FUNCTION_BLOCK CsvPersistantEventStorage IMPLEMENTS I_PersistentEventStorage
VAR
	fbFileOpen : FB_FileOpen := (sPathName := 'C:\Events.log', nMode := FOPEN_MODEAPPEND OR FOPEN_MODETEXT);
	fbFilePuts : FB_FilePuts;
	fbFileClose : FB_FileClose;
	eWriteState : (FILE_OPEN_TRIGGER,FILE_OPEN, WAIT_FOR_EVENT,WRITE_EVENT_TRIGGER, WRITE_EVENT, FILE_CLOSE_TRIGGER, FILE_CLOSE, ERROR);
	stEventWrittenToFile : ST_Event;
	CsvString: T_MaxString;
END_VAR

CASE eWriteState OF
	FILE_OPEN_TRIGGER :
		fbFileOpen(bExecute := TRUE);
		
	FILE_OPEN :
		fbFileOpen(bExecute := FALSE);
		IF fbFileOpen.bError THEN
			eWriteState := ERROR;
		ELSIF NOT fbFileOpen.bBusy AND fbFileOpen.hFile <> 0 THEN
			eWriteState := WAIT_FOR_EVENT;
		END_IF
		
	WAIT_FOR_EVENT : 
		// Do nothing
		
	WRITE_EVENT_TRIGGER : 
		CsvString := CreateCsvString(stEvent := stEventWrittenToFile);
		fbFilePuts(bExecute := TRUE,
			sLine := CsvString,
			hFile := fbFileOpen.hFile);
		eWriteState := WRITE_EVENT;
		
	WRITE_EVENT :
		fbFilePuts(bExecute := FALSE);
		IF fbFilePuts.bError THEN
			eWriteState := ERROR;
		ELSIF NOT fbFilePuts.bBusy THEN
			eWriteState := WAIT_FOR_EVENT;
		END_IF
		
	FILE_CLOSE_TRIGGER :
		fbFileClose(bExecute := TRUE,
			hFile := fbFileOpen.hFile);
		eWriteState := ERROR;
		
	FILE_CLOSE : 
		fbFileClose(bExecute := FALSE);
		IF fbFileClose.bError THEN
			eWriteState := ERROR;
		ELSIF fbFileClose.bBusy THEN
			eWriteState := FILE_OPEN_TRIGGER;
		END_IF
		
	ERROR:
		//Do nothing
END_CASE

METHOD PRIVATE CreateCsvString : T_MaxString
VAR_INPUT
	stEvent : REFERENCE TO ST_Event;
END_VAR
VAR
	TempString : T_MaxString;
END_VAR
TempString := TO_STRING(stEvent.eEventType);
TempString := CONCAT (STR1 := TempString, STR2 := ',');
TempString := CONCAT (STR1 := TempString, STR2 := TO_STRING(stEvent.eEventSeverity));
TempString := CONCAT (STR1 := TempString, STR2 := ',');
TempString := CONCAT (STR1 := TempString, STR2 := TO_STRING(stEvent.nEventIdentity));
TempString := CONCAT (STR1 := TempString, STR2 := ',');
TempString := CONCAT (STR1 := TempString, stEvent.sEventText);
TempString := CONCAT (STR1 := TempString, STR2 := ',');
TempString := CONCAT (STR1 := TempString, STR2 := TO_STRING (stEvent.dtTimestamp));
TempString := CONCAT (STR1 := TempString, STR2 := '$n'); // NewLine

CreateCsvString := TempString;
END_METHOD

{warning 'add method implementation '}
METHOD StoreEvent
VAR_INPUT
	stEvent	: ST_Event;
END_VAR
IF eWriteState = WAIT_FOR_EVENT THEN
	eWriteState := WRITE_EVENT;
END_IF
END_METHOD

END_FUNCTION_BLOCK

(* stored: Version 1.1.0.1, ProductVersion 3.1.4024.5
   POU CsvPersistantEventStorage: Id {7a2e0c5f-3324-46b7-9ddf-65afa5ad1eb1}, SpecialFunc None
   Method CreateCsvString: Id {e4742ac6-a8a0-4928-893e-0c7a58fa8969}
   Method StoreEvent: Id {630aae18-3f10-4750-a143-840eb3d056fe} *)
